FUNCTION_BLOCK ABSTRACT FB_AlarmBase IMPLEMENTS I_Alarm
VAR_OUTPUT
	bActive				: BOOL;
END_VAR
VAR
	iAlarmContext		: I_AlarmContext;
	nAlarmContextId		: DINT := ALARM_INVALID_CONTEXT_ID;
	nAlarmId			: DINT;
	fbActiveRTrig		: R_TRIG;
	fbActiveFTrig		: F_TRIG;
END_VAR

fbActiveRTrig(CLK := bActive);
fbActiveFTrig(CLK := bActive);

IF fbActiveRTrig.Q THEN
	CopyArgsToStack();
END_IF

IF bActive AND nAlarmContextId = ALARM_INVALID_CONTEXT_ID AND NOT iAlarmContext.IsAlarmBufferFull THEN
	// Add this alarm to alarm context
	nAlarmContextId := iAlarmContext.AddNewAlarm(THIS^);
END_IF

IF fbActiveFTrig.Q THEN
	IF nAlarmContextId <> ALARM_INVALID_CONTEXT_ID THEN
		// Prepare argument stack for new arguments
		ClearArgStack();
		// Remove this alarm from alarm context
		iAlarmContext.RemoveAlarm(nAlarmContextId);
		nAlarmContextId := ALARM_INVALID_CONTEXT_ID;
	END_IF
END_IF

PROPERTY AlarmId : DINT
GET
AlarmId := nAlarmId;
END_GET
END_PROPERTY

PROPERTY ABSTRACT ArgStackMemoryPointer : POINTER TO BYTE
GET
END_GET
END_PROPERTY

PROPERTY ABSTRACT ArgStackMemorySize : DINT
GET
END_GET
END_PROPERTY

METHOD PROTECTED ABSTRACT ClearArgStack
VAR_INPUT
END_VAR
END_METHOD

METHOD PROTECTED ABSTRACT CopyArgsToStack
VAR_INPUT
END_VAR
END_METHOD

METHOD FB_init : BOOL
VAR_INPUT
	bInitRetains		: BOOL; // if TRUE, the retain variables are initialized (warm start / cold start)
	bInCopyCode			: BOOL;  // if TRUE, the instance afterwards gets moved into the copy code (online change)
	iAlarmContext		: I_AlarmContext;
	nAlarmId			: DINT;
END_VAR
THIS^.iAlarmContext := iAlarmContext;
THIS^.nAlarmId := nAlarmId;
END_METHOD

END_FUNCTION_BLOCK

(* stored: Version 1.1.0.1, ProductVersion 3.1.4024.15
   POU FB_AlarmBase: Id {04313dcc-4e0a-48ee-b19d-8b92720ca9ef}, SpecialFunc None
   Property AlarmId: Id {2d1899b9-4017-4f95-8f6c-0034962310d9}
   Get Get: Id {4476556b-1d1a-477d-b3f1-647cdb1e10e5}
   Property ArgStackMemoryPointer: Id {0b0678ac-674b-42ea-a6dc-8513842eac7a}
   Get Get: Id {12a06311-a00e-467e-ae51-9be1c5db8ca7}
   Property ArgStackMemorySize: Id {7ca7e053-1df9-40d3-9e2c-a93e7fe96283}
   Get Get: Id {736a1dae-b3ea-4e72-9beb-06cfc93935c1}
   Method ClearArgStack: Id {15032434-4939-47dc-b1ee-cc562c777d55}
   Method CopyArgsToStack: Id {e4e54049-9092-4598-8c52-246ef39f02eb}
   Method FB_init: Id {5872302a-1c07-4ba2-b228-b76436212b67} *)
